FUNCTION_BLOCK CylinderBaseTestContext EXTENDS TcoCore._internals_TcoContext
VAR
	_sut			: CylinderBaseImplemented(THIS^);
	_sutInvalid		: CylinderBaseImplemented(THIS^);
	_atHomeSignal	: BOOL;	
	_atWorkSignal	: BOOL;	
	_toHomeSignal	: BOOL;	
	_toWorkSignal	: BOOL;
END_VAR
VAR
	_get_AtHome	: BOOL;
	_get_AtWork : BOOL;	
END_VAR

METHOD PROTECTED Main
_sut(inoAtHomePos := _atHomeSignal,
    inoAtWorkPos := _atWorkSignal,
    inoToHomePos := _toHomeSignal,
    inoToWorkPos := _toWorkSignal);
	
CASE _testId OF
	eCyclinderBaseTests.Invalid:
		_sutInvalid.AtHome;
		_sutInvalid.AtWork;
		_sutInvalid.Restore();
		_sutInvalid.Stop();
    eCyclinderBaseTests.GetAtHome:
		_get_AtHome := _sut.AtHome;		
    eCyclinderBaseTests.GetAtWork: 
		_get_AtWork := _sut.AtWork;               
END_CASE
END_METHOD

END_FUNCTION_BLOCK

(* stored: Version 1.1.0.1, ProductVersion 3.1.4024.9
   POU CylinderBaseTestContext: Id {e41369b8-4146-091a-3fca-553a7f936fbe}, SpecialFunc None
   Method Main: Id {db7fc157-6cb2-07ea-2d1f-c582b98c42b0} *)
